KUKA KRL program: testmod.src, testmod.dat

--- testmod.src ---
&ACCESS RV
DEF  testmod ( )
   ;FOLD INI;%{PE}
      ;FOLD BASISTECH INI
         GLOBAL INTERRUPT DECL 3 WHEN $STOPMESS==TRUE DO IR_STOPM ( )
         INTERRUPT ON 3
         BAS (#INITMOV,0 )
      ;ENDFOLD (BASISTECH INI)
      ;FOLD USER INI
         ;Make your modifications here

      ;ENDFOLD (USER INI)
   ;ENDFOLD (INI)

   ;FOLD PTP HOME  Vel= 100 % DEFAULT;%{PE}%MKUKATPBASIS,%CMOVE,%VPTP,%P 1:PTP, 2:HOME, 3:, 5:100, 7:DEFAULT
      $BWDSTART = FALSE
      PDAT_ACT=PDEFAULT
      FDAT_ACT=FHOME
      BAS (#PTP_PARAMS,100 )
      $H_POS=XHOME
      PTP  XHOME
   ;ENDFOLD

;fold HoldMyFoldyHolds
;endfold

;fold GripMyTerryFlaps
;endfold
;fold buttz
;endfold


   ;FOLD PTP HOME  Vel= 100 % DEFAULT;%{PE}%MKUKATPBASIS,%CMOVE,%VPTP,%P 1:PTP, 2:HOME, 3:, 5:100, 7:DEFAULT
      $BWDSTART = FALSE
      PDAT_ACT=PDEFAULT
      FDAT_ACT=FHOME
      BAS (#PTP_PARAMS,100 )
      $H_POS=XHOME
      PTP  XHOME
   ;ENDFOLD
END

--- testmod.dat ---
&ACCESS  RV
DEFDAT  testmod
;FOLD EXTERNAL DECLARATIONS;%{PE}%MKUKATPBASIS,%CEXT,%VCOMMON,%P
;FOLD BASISTECH EXT;%{PE}%MKUKATPBASIS,%CEXT,%VEXT,%P
EXT  BAS (BAS_COMMAND  :IN,REAL  :IN )
;ENDFOLD (BASISTECH EXT)
;FOLD USER EXT;%{E}%MKUKATPUSER,%CEXT,%VEXT,%P
;Make your modifications here

;ENDFOLD (USER EXT)
;ENDFOLD (EXTERNAL DECLARATIONS)
ENDDAT
